// TIA Portal project "Sorting_With_Hight" (V17)
// Vorlageprojekt für das Buch mit Zielsystem S7-1200

(* hardware
DEVICE "S7-1200-Station_1"  S7-1200 Station
   slot 0: "Baugruppenträger_0"  Rack  V1.0
   slot 1: "PLC_1"  CPU 1214C DC/DC/DC  6ES7 214-1AG40-0XB0  V4.5
*)

// ===== PLC "PLC_1"  CPU 1214C DC/DC/DC =====

VAR_GLOBAL   // PLC tag table "Standard-Variablentabelle"
   "High_Sensor" AT %I0.0 : Bool;
   "Low_sensor" AT %I0.1 : Bool;
   "Pallet_Sensor" AT %I0.2 : Bool;
   "Loaded_Sensor" AT %I0.3 : Bool;
   "Right_Entry_Sensor" AT %I0.4 : Bool;
   "Left_Entry_Sensor" AT %I0.5 : Bool;
   "Right_Exit_Sensor" AT %I0.6 : Bool;
   "Left_Exit_Sensor" AT %I0.7 : Bool;
   "Convayer_Entery" AT %Q0.0 : Bool;
   "Load" AT %Q0.1 : Bool;
   "Transfer_Right" AT %Q0.2 : Bool;
   "Transfer_Left" AT %Q0.3 : Bool;
   "Convayer_Right" AT %Q0.4 : Bool;
   "Convayer_Left" AT %Q0.5 : Bool;
   "Start" AT %I1.0 : Bool;
   "Reset" AT %I1.1 : Bool;
   "Stop" AT %I1.2 : Bool;
   "Load_Memory" AT %M0.0 : Bool;
   "High_Sensor_Memory" AT %M0.1 : Bool;
   "Low_Sensor_Memory" AT %M0.2 : Bool;
   "Convayer_Entery_Memory" AT %M0.3 : Bool;
   "System_Run_Memory" AT %M0.4 : Bool;
END_VAR

FUNCTION "MHJ-PLC-Lab-Function-S71200" : Void   // FC9000, SCL
{ S7_Optimized_Access := 'TRUE' }
VERSION : 0.1
   VAR_TEMP
      rdTimeReturn : Int;
      outputTime : DTL;
      SyncVal : Byte;
      forVal : Int;
      forVal_2 : Int;
      Value : Byte;
   END_VAR
   VAR CONSTANT
      CompVal : Byte := 16#34;
      Value_01 : Byte := 16#11;
      Value_01_DW : DWord := 16#A165_D992;
      Value_02_DW : DWord := 16#58BE_4401;
   END_VAR
BEGIN

   #Value:=PEEK(area := 16#82,
        dbNumber := 0,
        byteOffset := 511);
   #Value := #Value + 1;

   POKE(area := 16#82,
        dbNumber := 0,
        byteOffset := 511,
        value := #Value);

   POKE(area:=16#81,
        dbNumber:=0,
        byteOffset:=1016,
        value:=#Value_01_DW);
   POKE(area := 16#81,
        dbNumber := 0,
        byteOffset := 1020,
        value := #Value_02_DW);

   POKE(area := 16#81,
        dbNumber := 0,
        byteOffset := 511,
        value := B#16#00);

   FOR #forVal := 0 TO 120 DO
       FOR #forVal_2:=0 TO 10 DO
           #rdTimeReturn:=RD_SYS_T(#outputTime);
           #rdTimeReturn := WR_SYS_T(#outputTime);
           #rdTimeReturn := RD_SYS_T(#outputTime);
           #rdTimeReturn := WR_SYS_T(#outputTime);
       END_FOR;
       #SyncVal:= PEEK(area := 16#81,
                      dbNumber := 0,
                      byteOffset := 511);
       IF #SyncVal = #CompVal THEN
          GOTO M_1;
       END_IF;
   END_FOR;
   RETURN;

   M_1:
   POKE(area := 16#81,
        dbNumber := 0,
        byteOffset := 511,
        value := B#16#0);
END_FUNCTION

ORGANIZATION_BLOCK "Main"   // OB1, LAD, ProgramCycle
TITLE = "Main Program Sweep (Cycle)"
{ S7_Optimized_Access := 'TRUE' }
VERSION : 0.1
   VAR_INPUT
      Initial_Call : Bool;   // Initial call of this OB
      Remanence : Bool;   // =True, if remanent data are available
   END_VAR
BEGIN

REGION Network 1: Konnektierungsbaustein für PLC-Lab
   // Im Netzwerk 1 wird der Konnektierungsbaustein für PLC-Lab aufgerufen.
   // Dieser Aufruf darf nicht entfernt werden!
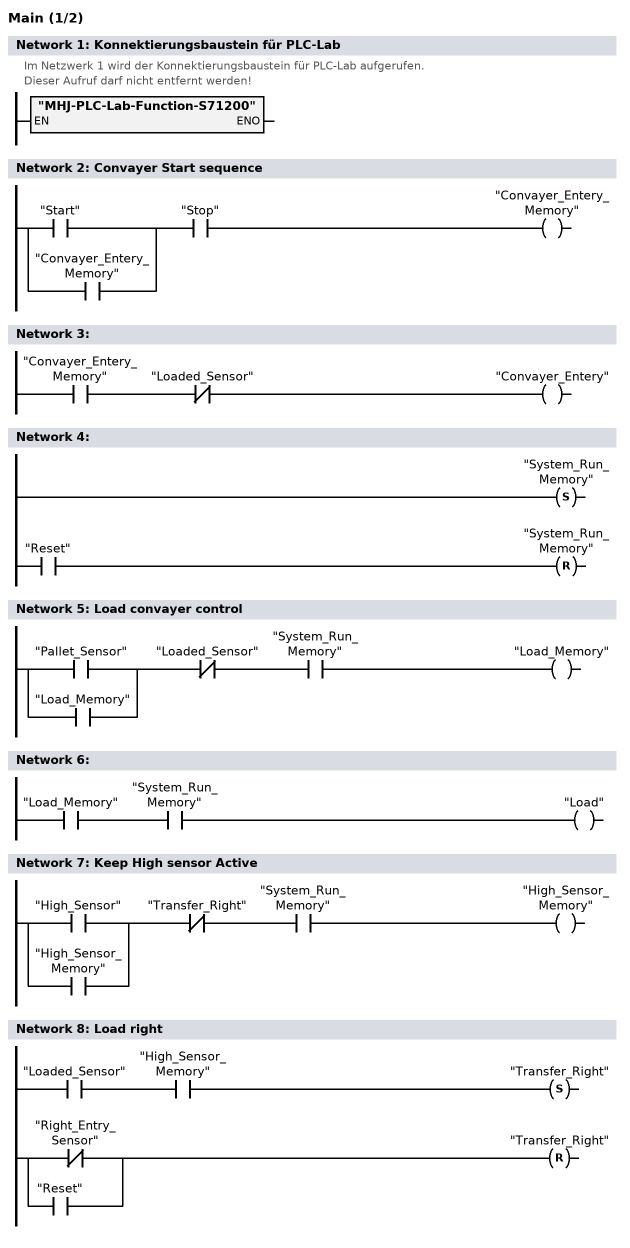
   RUNG wire#powerrail
      "MHJ-PLC-Lab-Function-S71200"()
   END_RUNG
   // the same network as SCL:
   "MHJ-PLC-Lab-Function-S71200"();
END_REGION

REGION Network 2: Convayer Start sequence
   RUNG wire#powerrail
      Contact( "Start" )
      wire#w1
      Contact( "Stop" )
      Coil( "Convayer_Entery_Memory" )
   END_RUNG
   RUNG wire#powerrail
      Contact( "Convayer_Entery_Memory" )
   END_RUNG wire#w1
   // the same network as SCL:
   "Convayer_Entery_Memory" := ("Start" OR "Convayer_Entery_Memory") AND "Stop";
END_REGION

REGION Network 3
   RUNG wire#powerrail
      Contact( "Convayer_Entery_Memory" )
      I_Contact( "Loaded_Sensor" )
      Coil( "Convayer_Entery" )
   END_RUNG
   // the same network as SCL:
   "Convayer_Entery" := "Convayer_Entery_Memory" AND NOT "Loaded_Sensor";
END_REGION

REGION Network 4
   RUNG wire#powerrail
      S_Coil( "System_Run_Memory" )
   END_RUNG
   RUNG wire#powerrail
      Contact( "Reset" )
      R_Coil( "System_Run_Memory" )
   END_RUNG
   // the same network as SCL:
   "System_Run_Memory" := TRUE;
   IF "Reset" THEN "System_Run_Memory" := FALSE; END_IF;
END_REGION

REGION Network 5: Load convayer control
   RUNG wire#powerrail
      Contact( "Pallet_Sensor" )
      wire#w1
      I_Contact( "Loaded_Sensor" )
      Contact( "System_Run_Memory" )
      Coil( "Load_Memory" )
   END_RUNG
   RUNG wire#powerrail
      Contact( "Load_Memory" )
   END_RUNG wire#w1
   // the same network as SCL:
   "Load_Memory" := ("Pallet_Sensor" OR "Load_Memory") AND NOT "Loaded_Sensor" AND "System_Run_Memory";
END_REGION

REGION Network 6
   RUNG wire#powerrail
      Contact( "Load_Memory" )
      Contact( "System_Run_Memory" )
      Coil( "Load" )
   END_RUNG
   // the same network as SCL:
   "Load" := "Load_Memory" AND "System_Run_Memory";
END_REGION

REGION Network 7: Keep High sensor Active
   RUNG wire#powerrail
      Contact( "High_Sensor" )
      wire#w1
      I_Contact( "Transfer_Right" )
      Contact( "System_Run_Memory" )
      Coil( "High_Sensor_Memory" )
   END_RUNG
   RUNG wire#powerrail
      Contact( "High_Sensor_Memory" )
   END_RUNG wire#w1
   // the same network as SCL:
   "High_Sensor_Memory" := ("High_Sensor" OR "High_Sensor_Memory") AND NOT "Transfer_Right" AND "System_Run_Memory";
END_REGION

REGION Network 8: Load right
   RUNG wire#powerrail
      Contact( "Loaded_Sensor" )
      Contact( "High_Sensor_Memory" )
      S_Coil( "Transfer_Right" )
   END_RUNG
   RUNG wire#powerrail
      I_Contact( "Right_Entry_Sensor" )
      wire#w1
      R_Coil( "Transfer_Right" )
   END_RUNG
   RUNG wire#powerrail
      Contact( "Reset" )
   END_RUNG wire#w1
   // the same network as SCL:
   IF "Loaded_Sensor" AND "High_Sensor_Memory" THEN "Transfer_Right" := TRUE; END_IF;
   IF NOT "Right_Entry_Sensor" OR "Reset" THEN "Transfer_Right" := FALSE; END_IF;
END_REGION

REGION Network 9: Convayer Right ON Latch
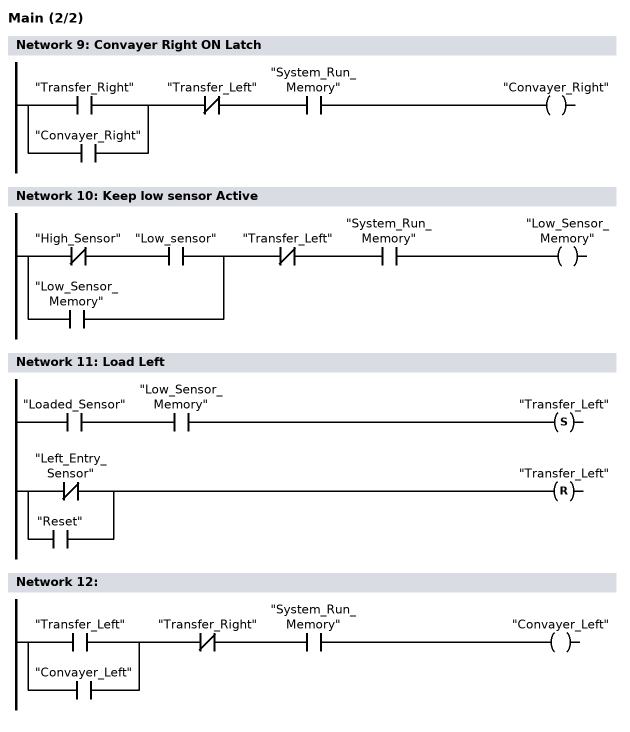
   RUNG wire#powerrail
      Contact( "Transfer_Right" )
      wire#w1
      I_Contact( "Transfer_Left" )
      Contact( "System_Run_Memory" )
      Coil( "Convayer_Right" )
   END_RUNG
   RUNG wire#powerrail
      Contact( "Convayer_Right" )
   END_RUNG wire#w1
   // the same network as SCL:
   "Convayer_Right" := ("Transfer_Right" OR "Convayer_Right") AND NOT "Transfer_Left" AND "System_Run_Memory";
END_REGION

REGION Network 10: Keep low sensor Active
   RUNG wire#powerrail
      I_Contact( "High_Sensor" )
      Contact( "Low_sensor" )
      wire#w1
      I_Contact( "Transfer_Left" )
      Contact( "System_Run_Memory" )
      Coil( "Low_Sensor_Memory" )
   END_RUNG
   RUNG wire#powerrail
      Contact( "Low_Sensor_Memory" )
   END_RUNG wire#w1
   // the same network as SCL:
   "Low_Sensor_Memory" := ((NOT "High_Sensor" AND "Low_sensor") OR "Low_Sensor_Memory") AND NOT "Transfer_Left" AND "System_Run_Memory";
END_REGION

REGION Network 11: Load Left
   RUNG wire#powerrail
      Contact( "Loaded_Sensor" )
      Contact( "Low_Sensor_Memory" )
      S_Coil( "Transfer_Left" )
   END_RUNG
   RUNG wire#powerrail
      I_Contact( "Left_Entry_Sensor" )
      wire#w1
      R_Coil( "Transfer_Left" )
   END_RUNG
   RUNG wire#powerrail
      Contact( "Reset" )
   END_RUNG wire#w1
   // the same network as SCL:
   IF "Loaded_Sensor" AND "Low_Sensor_Memory" THEN "Transfer_Left" := TRUE; END_IF;
   IF NOT "Left_Entry_Sensor" OR "Reset" THEN "Transfer_Left" := FALSE; END_IF;
END_REGION

REGION Network 12
   RUNG wire#powerrail
      Contact( "Transfer_Left" )
      wire#w1
      I_Contact( "Transfer_Right" )
      Contact( "System_Run_Memory" )
      Coil( "Convayer_Left" )
   END_RUNG
   RUNG wire#powerrail
      Contact( "Convayer_Left" )
   END_RUNG wire#w1
   // the same network as SCL:
   "Convayer_Left" := ("Transfer_Left" OR "Convayer_Left") AND NOT "Transfer_Right" AND "System_Run_Memory";
END_REGION
END_ORGANIZATION_BLOCK